(* IEC 61131-3 sources: robocpp/validation/corpus/regressions, 1 file *)

(* ---- array_repetition_count_limit.st ---- *)
(* validation: feature=regression.parser-array-repetition-limit clause=limits origin=seeded-limit *)
PROGRAM ArrayRepetitionCountLimit
VAR
    Motor : BOOL := [[00000000000000001629084365346150(096[[[[[[[[LSE;
END_VAR
END_PROGRAM
